{attribute 'GeneratedUsingTerminal: EPP5101-0002-0016'}
{attribute addProperty BoxType "EPP5101-0002-0016"}
{attribute addProperty Id "Enable_latch_CBOOL1Set_counterBOOL1"}
{attribute addProperty CRC "3573590905"}
{attribute addProperty Size "2"}
TYPE Control_D500AB79 :
STRUCT
	{attribute addProperty Name "Enable_latch_C"}
	Enable_latch_C : BOOL;
	{attribute addProperty Name "Set_counter"}
	Set_counter : BOOL;
END_STRUCT
END_TYPE

(* stored: Version 1.2.0.0, ProductVersion 3.1.4024.9
   DUT Control_D500AB79: Id {533f5555-ff89-480e-b0cc-7506e819285a} *)
